FUNCTION_BLOCK FB_Axis
(* 8888888888888888   SFC   8888888888888888888888*)
VAR_INPUT
	ResumeSFC             	: BOOL; 			(*	not automatic	*)
	ResetError            	: BOOL; 			(*	not automatic	*)
	fVelocity             	: LREAL := 20;
	sFB_Num				  	: STRING(3):='000'; // 3 digits for error list
	
	sFB_ModuleDescription 	: STRING(30):='';
	bPause				  	: BOOL;
	bReset				  	: BOOL;
	bModuloMode			  	: BOOL				:=FALSE;	
	eMotionType				: MC_MotionType		:=MC_MotionType.eAbsolute;
	eMotionDirection		: MC_Direction		:=MC_Direction.MC_Undefined_Direction;
	bTargetChanged			: BOOL;


END_VAR
VAR
	SFCCurrentStep      : STRING;
	SFCErrorPOU         : STRING;
	SFCErrorStep        : STRING;
	SFCError            : BOOL;
	SFCPause            : BOOL;
	SFCInit             : BOOL;
	SFCTipMode          : BOOL;
	SFCTip              : BOOL;
	SFCEnableLimit		: BOOL:=TRUE;
	// Reset Error
	SFCReset			: BOOL;
	ErrorSFC              : BOOL; 		(*	not automatic	*)
	Last_SFCErrorStep     : STRING; 	(*	not automatic	*)
	ErrorToPrint          : STRING; 	(*	not automatic	*)
	ton_SFCInit           : TON;
	ton_Disable           : TON;
	bMotionDone           : BOOL;
	ton_ResumeSFC_OffDelay: TON;
	sFB_ID                : STRING(4):='001';
	sActErrorID           : STRING(4);
	fbFormatString		  : FB_FORMATSTRING;
	sFullErrorId		  : STRING(12);//sAAAxBBBxEEE
	fb_SFC_Cycle		  : FB_SFC_Cycle;
	bNonPausedCycle: BOOL;
	rt_Resume: R_TRIG;

	iStepNo2: INT;
	iStepNo3: INT;
	ton_Delay: TON;
	bStepDone: BOOL;
	rt_TargetChanged: R_TRIG;
	op_Motor		: E_OperationButtons:=0;
END_VAR
(* 8888888888888888   END SFC   8888888888888888888888*)
VAR_INPUT
	bAutoDisable	: BOOL := FALSE;	(*	At not moving 30 sec	*)
	iAxisNum		: INT;
	fTollerance		: REAL:=0.1;
	fReference		: REAL:=0;
	bReadOffsetParameter   : BOOL;
	bWriteOffsetParameter  : BOOL;
	bSetZeroPB             : BOOL;
	fActPosSetToZero       : LREAL;
	
END_VAR
VAR_IN_OUT
	stOperation		: ST_OperationButtons;
	Points			: ST_AxisPoints;
	iTarget			: INT;
	iSubTarget		: INT;
END_VAR



VAR
	Shelf: INT;
	i				: INT;
	k				: INT;
	c_InPos			: INT;
	iLastTarget		: INT;
	iLastSubTarget	: INT;
	fLastPosition	: REAL;
	//sFB_Num         : STRING(3):='000';
	
	fbReadWrite_NC_PB  :FB_ReadWrite_NC_PB;
	iStepNo: INT;

END_VAR

VAR_OUTPUT
	fReadeToEncoderOffset  : LREAL;
END_VAR

VAR CONSTANT
	iStartPoint		: INT:=1;
	iPointNum		: INT:=15;
	iStartSubPoint	: INT:=-2;
	iSubPointNum	: INT:=2;
END_VAR

op_Motor:=stOperation.iActOperation;
act_InPosCalc();
act_GetErrorID();
act_Oper();
act_ReadWrite_NC_PB();
ton_ResumeSFC_OffDelay(PT:=T#0.1S);
rt_Resume(CLK:=stOperation.iActOperation=E_OperationButtons.ePlayAll);
rt_TargetChanged(CLK:=bTargetChanged);
IF rt_Resume.Q  THEN
	ton_ResumeSFC_OffDelay.IN:=TRUE;
END_IF
IF ton_ResumeSFC_OffDelay.Q THEN
	ton_ResumeSFC_OffDelay.IN:=FALSE;
	bNonPausedCycle:=FALSE;
	SFCPause:=FALSE;
	SFCError:=FALSE;
END_IF
IF stOperation.bStopResetAll THEN;
	stAxesfunctions[iAxisNum].bMcHalt:=FALSE;
	iSubTarget:=0;
	iTarget:=0;
END_IF
fb_SFC_Cycle
(
	sCycleName:= 'Axis Control', 
	bSFCError:=SFCError , //
	sSFCCurrentStep:=SFCCurrentStep , 
	sSFCErrorStep:= SFCErrorStep, 
	sSFCErrorPOU:=SFCErrorPOU , 
	sActErrorID:=sFullErrorId,
	//sFB_ModuleDescription:= CONCAT(sFB_ModuleDescription,INT_TO_STRING(iFB_Num)), 
	sFB_ModuleDescription:= sFB_ModuleDescription, 
	sLast_SFCErrorStep=>Last_SFCErrorStep , 
	bErrorSFC_Occured=> ErrorSFC, 
	//sErrorToPrint=>ErrorToPrint ,
	//sLast_ErrorToPrint=>, 
	bSFCInit=>SFCInit , 
	stOperation:=stOperation ,
	bResumeSFC:=ResumeSFC , 
	bResetError:=ResetError , 
	bSFCPause:=bNonPausedCycle,// SFCPause, bNonPausedCycle
	bResetCycle:=SFCReset
);


(*act_Locations;*)

ton_Disable(	PT:=T#30S,
			IN:=bAutoDisable
			AND stAxis[iAxisNum].Status.NotMoving
			AND stAxesfunctions[iAxisNum].McPowerState
			AND NOT stAxis[iAxisNum].Status.Disabled);

ACTION act_GetErrorID:
IF ErrorSFC THEN;
	// Initialization
	IF    Last_SFCErrorStep='MotorPowerNotOK' 		THEN sActErrorID:='001';
	ELSIF Last_SFCErrorStep='WatingMotionDone' 	    THEN sActErrorID:='002';
	ELSIF Last_SFCErrorStep='InPosCheck_1' 		    THEN sActErrorID:='003';
	ELSIF Last_SFCErrorStep='LimitDetected'         THEN sActErrorID:='004';
	ELSIF Last_SFCErrorStep='StopAxis'         		THEN sActErrorID:='005';	
	ELSE
		 sActErrorID:='999';
	END_IF
	
//ELSIF bWarning THEN;
	// Leave the warning message to print
ELSE;
		 sActErrorID:='000';
END_IF




fbFormatString(
	sFormat:= '%.3sx%.3sx%.3s', 
	arg1:= F_STRINGEx(sFB_ID), 
	arg2:= F_STRINGEx(sFB_Num), 
	arg3:= F_STRINGEx(sActErrorID), 
	sOut=>sFullErrorId );
	
//(*Clean Last ErrID*)IF NOT SFCPause AND NOT ErrorSFC THEN	sFullErrorId:='';END_IF
END_ACTION

ACTION act_InPosCalc:
;
k:=0;
FOR i:=iStartPoint TO iPointNum DO
	FOR k:=iStartSubPoint TO iSubPointNum DO
		Points.arInPos[i,k]:=FALSE;
	END_FOR
END_FOR


FOR i:=iStartPoint TO iPointNum DO
	FOR k:=iStartSubPoint TO iSubPointNum DO
		IF 	(NOT bModuloMode)
		AND eMotionType=MC_MotionType.eAbsolute
		AND stAxis[iAxisNum].NcToPlc.ActPos > Points.arPos[i,k]-fTollerance
		AND stAxis[iAxisNum].NcToPlc.ActPos < Points.arPos[i,k]+fTollerance
		AND stAxis[iAxisNum].Status.NotMoving
		(*AND stAxis[iAxisNum].Status.StandStill*)
		AND stAxis[iAxisNum].Status.InTargetPosition	THEN
			Points.arInPos[i,k]:=TRUE;
		ELSIF bModuloMode
		AND eMotionType=MC_MotionType.eAbsolute
		AND stAxis[iAxisNum].NcToPlc.ModuloActPos > Points.arPos[i,k]-fTollerance
		AND stAxis[iAxisNum].NcToPlc.ModuloActPos < Points.arPos[i,k]+fTollerance
		AND stAxis[iAxisNum].Status.NotMoving
		(*AND stAxis[iAxisNum].Status.StandStill*)
		AND stAxis[iAxisNum].Status.InTargetPosition	THEN
			Points.arInPos[i,k]:=TRUE;			
		END_IF
	END_FOR
END_FOR


c_InPos:=0;
FOR i:=iStartPoint TO iPointNum DO
	FOR k:=iStartSubPoint TO iSubPointNum DO
		IF Points.arInPos[i,k] THEN
			c_InPos:=c_InPos+1;
		END_IF
	END_FOR
END_FOR
END_ACTION

ACTION act_Oper:
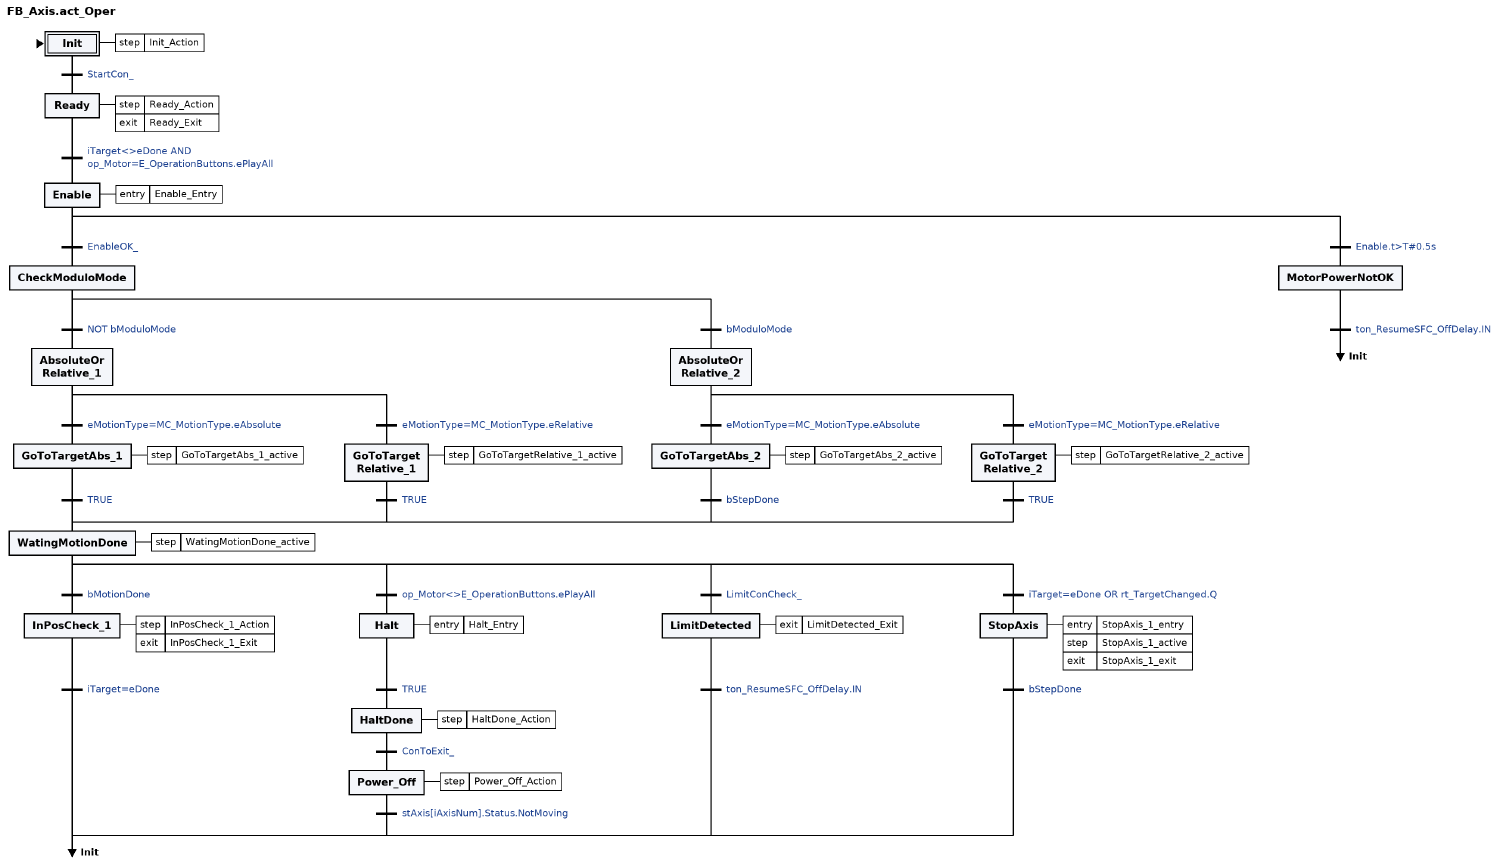
INITIAL_STEP Init:  // min time T#30ms
    Init_Action(N);  // step action
END_STEP
TRANSITION FROM Init TO Ready
    := StartCon_;
END_TRANSITION
STEP Ready:  // min time T#50ms
    Ready_Action(N);  // step action
    Ready_Exit(P0);  // exit action
END_STEP
TRANSITION FROM Ready TO Enable
    := iTarget<>eDone AND op_Motor=E_OperationButtons.ePlayAll;
END_TRANSITION
STEP Enable:
    Enable_Entry(P1);  // entry action
END_STEP
TRANSITION FROM Enable TO CheckModuloMode
    := EnableOK_;
END_TRANSITION
STEP CheckModuloMode:
END_STEP
TRANSITION FROM CheckModuloMode TO AbsoluteOrRelative_1
    := NOT bModuloMode;
END_TRANSITION
STEP AbsoluteOrRelative_1:
END_STEP
TRANSITION FROM AbsoluteOrRelative_1 TO GoToTargetAbs_1
    := eMotionType=MC_MotionType.eAbsolute;
END_TRANSITION
STEP GoToTargetAbs_1:  // min time T#0.1S, max time T#90S
    GoToTargetAbs_1_active(N);  // step action
END_STEP
TRANSITION FROM GoToTargetAbs_1 TO WatingMotionDone
    := TRUE;
END_TRANSITION
TRANSITION FROM AbsoluteOrRelative_1 TO GoToTargetRelative_1
    := eMotionType=MC_MotionType.eRelative;
END_TRANSITION
STEP GoToTargetRelative_1:  // min time T#0.1S, max time T#90S
    GoToTargetRelative_1_active(N);  // step action
END_STEP
TRANSITION FROM GoToTargetRelative_1 TO WatingMotionDone
    := TRUE;
END_TRANSITION
TRANSITION FROM CheckModuloMode TO AbsoluteOrRelative_2
    := bModuloMode;
END_TRANSITION
STEP AbsoluteOrRelative_2:
END_STEP
TRANSITION FROM AbsoluteOrRelative_2 TO GoToTargetAbs_2
    := eMotionType=MC_MotionType.eAbsolute;
END_TRANSITION
STEP GoToTargetAbs_2:  // min time T#0.1S, max time T#90S
    GoToTargetAbs_2_active(N);  // step action
END_STEP
TRANSITION FROM GoToTargetAbs_2 TO WatingMotionDone
    := bStepDone;
END_TRANSITION
TRANSITION FROM AbsoluteOrRelative_2 TO GoToTargetRelative_2
    := eMotionType=MC_MotionType.eRelative;
END_TRANSITION
STEP GoToTargetRelative_2:  // min time T#0.1S, max time T#90S
    GoToTargetRelative_2_active(N);  // step action
END_STEP
TRANSITION FROM GoToTargetRelative_2 TO WatingMotionDone
    := TRUE;
END_TRANSITION
TRANSITION FROM Enable TO MotorPowerNotOK
    := Enable.t>T#0.5s;
END_TRANSITION
STEP MotorPowerNotOK:  // max time T#100MS
END_STEP
TRANSITION FROM MotorPowerNotOK TO Init
    := ton_ResumeSFC_OffDelay.IN;
END_TRANSITION
STEP WatingMotionDone:
    WatingMotionDone_active(N);  // step action
END_STEP
TRANSITION FROM WatingMotionDone TO InPosCheck_1
    := bMotionDone;
END_TRANSITION
STEP InPosCheck_1:  // max time T#50ms
    InPosCheck_1_Action(N);  // step action
    InPosCheck_1_Exit(P0);  // exit action
END_STEP
TRANSITION FROM InPosCheck_1 TO Init
    := iTarget=eDone;
END_TRANSITION
TRANSITION FROM WatingMotionDone TO Halt
    := op_Motor<>E_OperationButtons.ePlayAll;
END_TRANSITION
STEP Halt:  // min time T#1S
    Halt_Entry(P1);  // entry action
END_STEP
TRANSITION FROM Halt TO HaltDone
    := TRUE;
END_TRANSITION
STEP HaltDone:
    HaltDone_Action(N);  // step action
END_STEP
TRANSITION FROM HaltDone TO Power_Off
    := ConToExit_;
END_TRANSITION
STEP Power_Off:
    Power_Off_Action(N);  // step action
END_STEP
TRANSITION FROM Power_Off TO Init
    := stAxis[iAxisNum].Status.NotMoving;
END_TRANSITION
TRANSITION FROM WatingMotionDone TO LimitDetected
    := LimitConCheck_;
END_TRANSITION
STEP LimitDetected:  // max time T#100MS
    LimitDetected_Exit(P0);  // exit action
END_STEP
TRANSITION FROM LimitDetected TO Init
    := ton_ResumeSFC_OffDelay.IN;
END_TRANSITION
TRANSITION FROM WatingMotionDone TO StopAxis
    := iTarget=eDone OR rt_TargetChanged.Q;
END_TRANSITION
STEP StopAxis:  // max time T#5s
    StopAxis_1_entry(P1);  // entry action
    StopAxis_1_active(N);  // step action
    StopAxis_1_exit(P0);  // exit action
END_STEP
TRANSITION FROM StopAxis TO Init
    := bStepDone;
END_TRANSITION
// branch label Branch1_act_Oper
// branch label Branch0_act_Oper
END_ACTION

ACTION act_ReadWrite_NC_PB:
ton_Delay();
IF iAxisNum>0 AND iAxisNum<=C_Max_AxesCount THEN;
	fbReadWrite_NC_PB
	(
		bReadParameter:= , 
		bWriteParameter:= , 	
		iAxisNum:=iAxisNum , 
		mcAxisParameter:=MC_AxisParameter.AxisEncoderOffset , 	 
		bReatBusy=> , 
		bWriteBusy=> , 
		bReatError=> , 
		bWriteError=> ,
		fReadEncoderOffset=>,
		fWriteEncoderOffset:=ar_AxisPos_BIOS[iAxisNum]		
		);


	IF bReadOffsetParameter THEN
			CASE iStepNo OF
			0:
			  fbReadWrite_NC_PB.iAxisNum := iAxisNum ;
			  fReadeToEncoderOffset:=0;
			  iStepNo :=10;
			  
		   10:
			  IF NOT fbReadWrite_NC_PB.bReatBusy AND NOT fbReadWrite_NC_PB.bReatError THEN
				 fbReadWrite_NC_PB.bReadParameter := TRUE;
				 iStepNo :=20;
			  END_IF
			  
		   20:
			 IF fbReadWrite_NC_PB.bReatBusy AND NOT fbReadWrite_NC_PB.bReatError THEN
				fbReadWrite_NC_PB.bReadParameter := FALSE;
				iStepNo :=30; 
			   END_IF
			   
			30:
			   fReadeToEncoderOffset:= fbReadWrite_NC_PB.fReadEncoderOffset;
			   ar_AxisPos_BIOS[iAxisNum]:= fbReadWrite_NC_PB.fReadEncoderOffset;
			   bReadOffsetParameter := FALSE;
			   iStepNo :=0;
	
			END_CASE
	END_IF
	
	(*********************** Write Offset *************************)
	
	IF bWriteOffsetParameter THEN
			CASE iStepNo2 OF
				
			0:
			  fbReadWrite_NC_PB.iAxisNum := iAxisNum ;
			  stAxesfunctions[iAxisNum].bMcPower:=FALSE;
			  ton_Delay.PT:=T#0.5S;ton_Delay.IN:=TRUE;			  
			  iStepNo2 :=5;
			5:IF ton_Delay.Q THEN;
				 iStepNo2 :=10;
				 ton_Delay.IN:=FALSE;
			  END_IF
			  
		   10:
			  IF NOT fbReadWrite_NC_PB.bWriteBusy AND NOT fbReadWrite_NC_PB.bWriteError THEN
				 fbReadWrite_NC_PB.bWriteParameter := TRUE;
				 iStepNo2 :=20;
			  END_IF
			  
		   20:
			 IF fbReadWrite_NC_PB.bWriteBusy AND NOT fbReadWrite_NC_PB.bWriteError THEN
				fbReadWrite_NC_PB.bWriteParameter := FALSE;
				iStepNo2 :=30; 
			   END_IF
			   
			30:
			   bWriteOffsetParameter  := FALSE;
			   bReadOffsetParameter:=TRUE;
			   iStepNo2 :=0;
			END_CASE
	END_IF
	
	
	
	(************************* Set Zero ****************************)
	
	IF bSetZeroPB THEN
		CASE iStepNo3 OF
			
		   0:
			 fActPosSetToZero := stAxis[iAxisNum].NcToPlc.ActPos - fReadeToEncoderOffset;
			 ar_AxisPos_BIOS[iAxisNum] := fActPosSetToZero * -1;
			 iStepNo3 :=10;
		  10:
			 bWriteOffsetParameter := TRUE;
			 iStepNo3 :=20;
		  20:
			 bSetZeroPB := FALSE;
			 iStepNo3 :=0;
	
		END_CASE
	END_IF

END_IF
END_ACTION

TRANSITION ConToExit_:
stAxesfunctions[iAxisNum].McHaltDone
OR
stAxesfunctions[iAxisNum].McStopDone
OR
(NOT stAxis[iAxisNum].Status.Stopping)
END_TRANSITION

ACTION Enable_Entry:
stAxesfunctions[iAxisNum].bMcPower:=TRUE;
END_ACTION

TRANSITION EnableOK_:
stAxesfunctions[iAxisNum].McPowerState
AND
stAxesfunctions[iAxisNum].bAxReleaseNeg
AND
stAxesfunctions[iAxisNum].bAxReleasePos
END_TRANSITION

ACTION GoToTargetAbs_1_active:
IF iTarget<>0 AND iTarget<=iPointNum AND iTarget>=iStartPoint THEN
	stAxesfunctions[iAxisNum].fPosition:=Points.arPos[iTarget,iSubTarget];
	fLastPosition:=Points.arPos[iTarget,iSubTarget];
	iLastTarget:=iTarget;
	iLastSubTarget:=iSubTarget;
END_IF

IF stAxesfunctions[iAxisNum].fPosition=Points.arPos[iTarget,iSubTarget] THEN
	stAxesfunctions[iAxisNum].fVelocity:=fVelocity;
	stAxesfunctions[iAxisNum].bMcMoveAbs:=TRUE;
	stAxesfunctions[iAxisNum].bMcHalt:=FALSE;
END_IF
END_ACTION

ACTION GoToTargetAbs_2_active:
IF iTarget<>0 AND iTarget<=iPointNum AND iTarget>=iStartPoint THEN
	stAxesfunctions[iAxisNum].fPosition:=Points.arPos[iTarget,iSubTarget];
	fLastPosition:=Points.arPos[iTarget,iSubTarget];
	iLastTarget:=iTarget;
	iLastSubTarget:=iSubTarget;
END_IF

IF stAxesfunctions[iAxisNum].fPosition=Points.arPos[iTarget,iSubTarget] THEN
	stAxesfunctions[iAxisNum].fVelocity:=fVelocity;
	stAxesfunctions[iAxisNum].iDirection:=eMotionDirection;
	stAxesfunctions[iAxisNum].bMcHalt:=FALSE;		
	IF eMotionDirection=MC_Direction.MC_Positive_Direction OR eMotionDirection=MC_Direction.MC_Negative_Direction THEN;
		IF ABS(stAxesfunctions[iAxisNum].fPosition-stAxis[iAxisNum].NcToPlc.ModuloActPos)<30
		OR ABS(stAxesfunctions[iAxisNum].fPosition-stAxis[iAxisNum].NcToPlc.ModuloActPos)>330
		THEN;
			stAxesfunctions[iAxisNum].iDirection:=MC_Direction.MC_Shortest_Way;
			stAxesfunctions[iAxisNum].bMcMoveModulo:=TRUE;
			bStepDone:=TRUE;
		ELSE;
			stAxesfunctions[iAxisNum].bMcMoveModulo:=TRUE;
			bStepDone:=TRUE;
		END_IF
	ELSIF eMotionDirection=MC_Direction.MC_Shortest_Way THEN;
		stAxesfunctions[iAxisNum].bMcMoveModulo:=TRUE;
		bStepDone:=TRUE;
	ELSE
		bStepDone:=FALSE;		
	END_IF
ELSE
	bStepDone:=FALSE;
END_IF
END_ACTION

ACTION GoToTargetRelative_1_active:

END_ACTION

ACTION GoToTargetRelative_2_active:

END_ACTION

ACTION Halt_Entry:
	stAxesfunctions[iAxisNum].bMcMoveAbs:=FALSE;
	stAxesfunctions[iAxisNum].bMcMoveRel:=FALSE;
	stAxesfunctions[iAxisNum].bMcMoveModulo:=FALSE;
	stAxesfunctions[iAxisNum].bMcHalt:=TRUE;
	iTarget:=0;
END_ACTION

ACTION HaltDone_Action:
IF 	stAxesfunctions[iAxisNum].McHaltErr THEN
	stAxesfunctions[iAxisNum].bMcStop:=TRUE;
END_IF
END_ACTION

ACTION Init_Action:
stAxesfunctions[iAxisNum].bMcMoveAbs:=FALSE;
stAxesfunctions[iAxisNum].bMcMoveRel:=FALSE;
stAxesfunctions[iAxisNum].bMcMoveModulo:=FALSE;
//stAxesfunctions[iAxisNum].bMcHalt:=FALSE;
stAxesfunctions[iAxisNum].fAcceleration:=0;
stAxesfunctions[iAxisNum].fDeceleration:=0;
stAxesfunctions[iAxisNum].fJerk:=0;
SFCReset:=FALSE;
bTargetChanged:=FALSE;
END_ACTION

ACTION InPosCheck_1_Action:
IF iTarget >=iStartPoint AND iTarget<=iPointNum THEN
	IF Points.arInPos[iTarget,iSubTarget]
	AND stAxis[iAxisNum].Status.InTargetPosition
	//AND stAxesfunctions[iAxisNum].McMoveAbsoluteDone  
	THEN;
		iTarget:=eDone;
		iSubTarget:=eDone;
	END_IF
END_IF
END_ACTION

ACTION InPosCheck_1_Exit:
stAxesfunctions[iAxisNum].bMcMoveAbs:=FALSE;
stAxesfunctions[iAxisNum].bMcMoveRel:=FALSE;
stAxesfunctions[iAxisNum].bMcMoveModulo:=FALSE;
//bMotionDone:=TRUE;
END_ACTION

TRANSITION LimitConCheck_:
NOT stAxesfunctions[iAxisNum].McPowerState
OR
NOT stAxesfunctions[iAxisNum].bAxReleaseNeg
OR
NOT stAxesfunctions[iAxisNum].bAxReleasePos
END_TRANSITION

ACTION LimitDetected_Exit:
SFCReset:=TRUE;
END_ACTION

TRANSITION NoReq_:
iTarget=eDone
END_TRANSITION

TRANSITION NoReq__1:
iTarget=eDone
END_TRANSITION

ACTION Power_Off_Action:
IF NOT stAxis[iAxisNum].Status.NotMoving THEN
	stAxesfunctions[iAxisNum].bMcPower:=FALSE;
END_IF
END_ACTION

ACTION Ready_Action:
IF 	stAxesfunctions[iAxisNum].bMcHalt AND op_Motor=E_OperationButtons.ePlayAll THEN;
	iSubTarget:=iLastSubTarget;
	iTarget:=iLastTarget;
END_IF


IF ton_Disable.Q THEN
	stAxesfunctions[iAxisNum].bMcPower:=FALSE;
END_IF
END_ACTION

ACTION Ready_Exit:
bMotionDone:=FALSE;
stAxesfunctions[iAxisNum].bMcStop:=FALSE;
END_ACTION

TRANSITION StartCon_:
NOT stAxesfunctions[iAxisNum].McMoveAbsoluteDone
AND
NOT stAxesfunctions[iAxisNum].bMcMoveAbs
END_TRANSITION

ACTION StopAxis_1_active:
IF stAxesfunctions[iAxisNum].McStopDone THEN;
	bStepDone:=TRUE;
ELSE;
	bStepDone:=FALSE;
END_IF
END_ACTION

ACTION StopAxis_1_entry:
	stAxesfunctions[iAxisNum].bMcMoveAbs:=FALSE;
	stAxesfunctions[iAxisNum].bMcMoveRel:=FALSE;
	stAxesfunctions[iAxisNum].bMcMoveModulo:=FALSE;
	
	stAxesfunctions[iAxisNum].bMcStop:=TRUE;
END_ACTION

ACTION StopAxis_1_exit:
stAxesfunctions[iAxisNum].bMcStop:=FALSE;
END_ACTION

ACTION WatingMotionDone_active:
bMotionDone:=FALSE;
IF bModuloMode THEN;
	IF eMotionType=MC_MotionType.eAbsolute
	AND stAxesfunctions[iAxisNum].McMoveModuloDone
	THEN;
		bMotionDone:=TRUE;
	ELSIF eMotionType=MC_MotionType.eRelative 
	AND FALSE	
	THEN;
		bMotionDone:=TRUE;
	ELSE;
		bMotionDone:=FALSE;
	END_IF
ELSE;
	IF eMotionType=MC_MotionType.eAbsolute 
	AND stAxesfunctions[iAxisNum].McMoveAbsoluteDone
	THEN;
		bMotionDone:=TRUE;
	ELSIF eMotionType=MC_MotionType.eRelative
 	AND FALSE
	THEN;
		bMotionDone:=TRUE;
	ELSE;
		bMotionDone:=FALSE;
	END_IF	
END_IF
END_ACTION

END_FUNCTION_BLOCK

(* stored: Version 1.1.0.1, ProductVersion 3.1.4024.12
   POU FB_Axis: Id {bc990690-b581-413e-b58e-2a5ff921a80a}, SpecialFunc None
   Folder Actions: Id {19a40766-b7eb-4c73-a4d3-090adc0dc6ee}
   Folder Trans: Id {2a0730e9-7a28-47d9-8b64-35e038d1884f}
   Action act_GetErrorID: Id {c7fcb077-28ef-481e-8b12-2903faa42a79}
   Action act_InPosCalc: Id {6d22facd-de77-446f-8756-a5b8b563146e}
   Action act_Oper: Id {ef55d58b-7fe3-418a-bc82-973ba88b2a05}
   Action act_ReadWrite_NC_PB: Id {77dcfb9e-0415-4be2-a549-f01ba5e38427}
   Transition ConToExit_: Id {8b0a15dd-fd97-405f-a3c0-8e30f6d5a021}
   Action Enable_Entry: Id {790b1e52-2418-455b-bed0-0ee6632b9fc4}
   Transition EnableOK_: Id {20fbcc47-66f5-4dd2-8a34-87b816e9331c}
   Action GoToTargetAbs_1_active: Id {ea89b8ee-7b6d-4e1a-87c8-1fd9e51c12ad}
   Action GoToTargetAbs_2_active: Id {8e292382-54f4-4305-b635-89f6c9bf316a}
   Action GoToTargetRelative_1_active: Id {ea19668a-110a-47a6-b5fe-b463696d0577}
   Action GoToTargetRelative_2_active: Id {d4de4710-f997-4e2f-9dd5-20d939f59bf5}
   Action Halt_Entry: Id {c3e8f353-c31d-4843-a7cd-1d8d8574a80a}
   Action HaltDone_Action: Id {ae5f33e7-5ac6-4693-be48-25885c105c7b}
   Action Init_Action: Id {0157bdc7-0271-4a2c-8c9d-e1bd1ae3210d}
   Action InPosCheck_1_Action: Id {61d4f6ab-80ff-4a16-a37e-d964c49bb924}
   Action InPosCheck_1_Exit: Id {512f78aa-a2dd-4891-a218-c5d498886451}
   Transition LimitConCheck_: Id {cb06290a-35e6-4fa6-beae-cc0811043341}
   Action LimitDetected_Exit: Id {9f8cda0c-d447-4fdd-8f3c-b5a5758479af}
   Transition NoReq_: Id {3b8d3037-1ce0-4f71-af7f-e5253891fcd7}
   Transition NoReq__1: Id {cf1ef19d-8947-4bcf-a011-68504d3c686c}
   Action Power_Off_Action: Id {654f985a-7d1b-422b-853d-e51d54419cf3}
   Action Ready_Action: Id {026512fd-0aaf-4545-803f-f74333f2b32f}
   Action Ready_Exit: Id {92c55298-2029-4089-a970-94edeb495178}
   Transition StartCon_: Id {02d178bf-84be-46a4-b531-c86bc3ffb92d}
   Action StopAxis_1_active: Id {90eafc07-383d-458e-bf5b-b6eb07e01600}
   Action StopAxis_1_entry: Id {34dda2c1-f9e9-4fce-8c49-6f0779e596c9}
   Action StopAxis_1_exit: Id {642e680b-77ff-468b-b48d-448b34bdc2ab}
   Action WatingMotionDone_active: Id {9e0deedb-8a54-4f99-a3a2-857490ae2ee2} *)
